// Examples of plant controlling.
// [Hint]
// > All reference-variables are implemented to ease monitoring of relevant variables.
FUNCTION_BLOCK FB_Plt_PlantControl EXTENDS FB_BA_View
VAR
   	{region 'Aggregates'}
		DmprSu_Open							: REFERENCE TO BOOL							REF= DmprSu.bOpen;
		DmprSu_Val							: REFERENCE TO REAL							REF= DmprSu.fActiveVal;
		DmprSu								: FB_TimerAggregateA						:= (iParent:=THIS^,					iLabel:=MyLabels.DmprSu);
		FanSu_Val							: REFERENCE TO UDINT						REF= FanSu.nActiveVal;
		FanSu								: FB_BA_AggregateM							:= (iParent:=THIS^,					iLabel:=MyLabels.FanSu);
			 
		DmprEx_Open							: REFERENCE TO BOOL							REF= DmprEx.bOpen;
		DmprEx_Val							: REFERENCE TO REAL							REF= DmprEx.fActiveVal;
		DmprEx								: FB_TimerAggregateA						:= (iParent:=THIS^,					iLabel:=MyLabels.DmprEx);
		FanEx_Val							: REFERENCE TO UDINT						REF= FanEx.nActiveVal;
		FanEx								: FB_BA_AggregateM							:= (iParent:=THIS^,					iLabel:=MyLabels.FanEx);
			 
		PreHtr_Proc							: REFERENCE TO BOOL							REF= PreHtr.Process.bActive;
		PreHtr_Val							: REFERENCE TO BOOL							REF= PreHtr.bActiveVal;
		PreHtr								: FB_ProcAggregateB							:= (iParent:=THIS^,					iLabel:=MyLabels.PreHtr,			Process:=(iLabel:=MyLabels.ProcPreRinse));
		Erc_Val								: REFERENCE TO BOOL							REF= Erc.bActiveVal;
		Erc									: FB_BA_AggregateB							:= (iParent:=THIS^,					iLabel:=MyLabels.Erc);
		Col_Val								: REFERENCE TO BOOL							REF= Col.bActiveVal;
		Col									: FB_BA_AggregateB							:= (iParent:=THIS^,					iLabel:=MyLabels.Col);
	{endregion}
	{region 'Plant'} 
		OpMode								: E_OpMod_AC								:= E_OpMod_AC.eOff;
		PlantCtrl_OpSta						: REFERENCE TO BOOL							REF= PlantCtrl.bOpSta;
		PlantCtrl_On						: REFERENCE TO BOOL							REF= PlantCtrl.bOn;
		PlantCtrl_PrVal						: REFERENCE TO UDINT						REF= PlantCtrl.nPresentValue;
		PlantCtrl_Step						: REFERENCE TO STRING						REF= PlantCtrl.sStep;
		PlantCtrl							: FB_BA_PlantCtrl := (
												iParent									:= THIS^,
												aOperationMode							:= [ E_OpMod_AC.eDisturb,			E_OpMod_AC.eSmokeExtract,		E_OpMod_AC.eOff,			E_OpMod_AC.eOn,				E_OpMod_AC.eNightCool ],
												aPriority								:= [ E_BA_Priority.eCritical,		E_BA_Priority.eLifeSafety,		E_BA_Priority.eProgram,		E_BA_Priority.eProgram,		E_BA_Priority.eProgram ],
												aAggregates := [(
													iReference							:= DmprSu,
													aOpMode								:= [ 0,								100,							0,							100,						100 ]
												), (
													iReference							:= DmprEx,
													aOpMode								:= [ 0,								100,							0,							100,						100 ]
												), (
													iReference							:= PreHtr,
													aOpMode								:= [ E_OpMod_Binary.eOff,			E_OpMod_Binary.eOn,				E_OpMod_Binary.eOff,		E_OpMod_Binary.eOn,			E_OpMod_Binary.eOff ],
													bWaitForProcesses					:= TRUE
												), (
													iReference							:= Erc,
													aOpMode								:= [ E_OpMod_Binary.eOff,			E_OpMod_Binary.eOn,				E_OpMod_Binary.eOff,		E_OpMod_Binary.eOn,			E_OpMod_Binary.eOff ]
												), (
													iReference							:= Col,
													aOpMode								:= [ E_OpMod_Binary.eOff,			E_OpMod_Binary.eOn,				E_OpMod_Binary.eOff,		E_OpMod_Binary.eOn,			E_OpMod_Binary.eOff ]
												), (
													iReference							:= FanSu,
													aOpMode								:= [ E_OpMod_Step2.eOff,			E_OpMod_Step2.eStep2,			E_OpMod_Step2.eOff,			E_OpMod_Step2.eStep1,		E_OpMod_Step2.eStep2 ],
													tDelayStepDown						:= T#0S,
													tDelayStepUp						:= T#5S
												), (
													iReference							:= FanEx,
													aOpMode								:= [ E_OpMod_Step2.eOff,			E_OpMod_Step2.eStep2,			E_OpMod_Step2.eOff,			E_OpMod_Step2.eStep1,		E_OpMod_Step2.eStep2 ],
													tDelayStepDown						:= T#5S,
													tDelayStepUp						:= T#0S
												)]
											);
	{endregion}
END_VAR

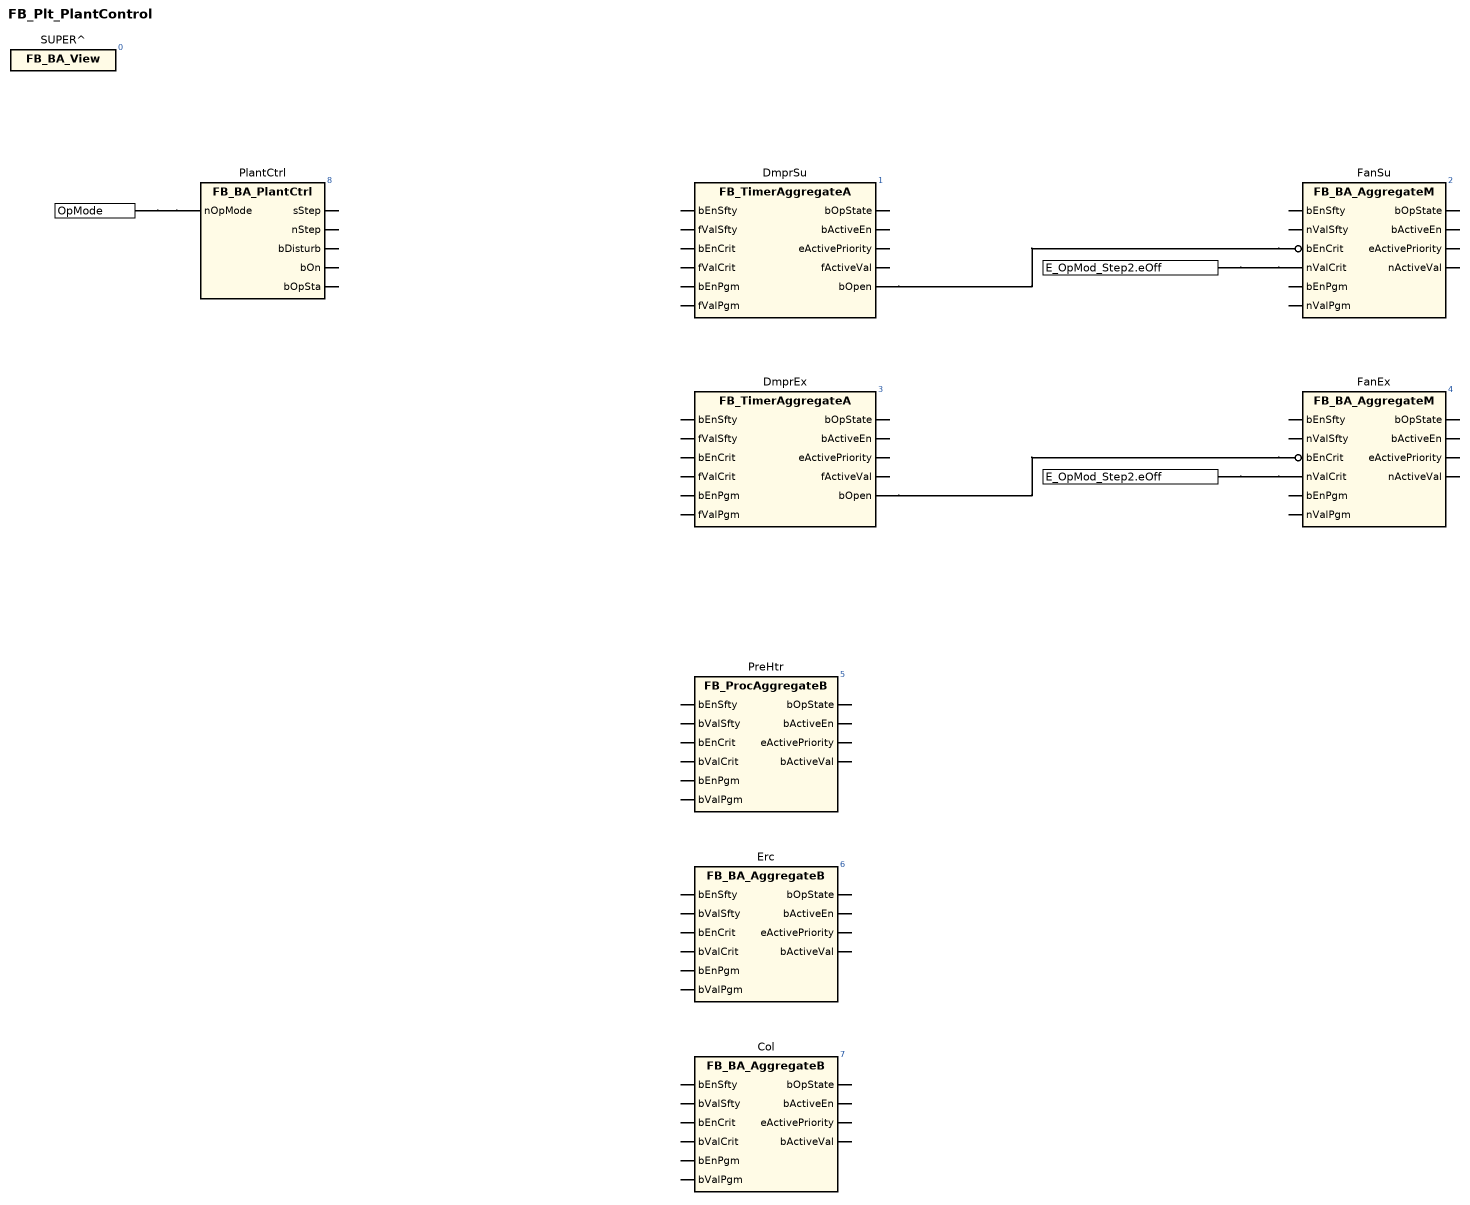
SUPER^(); // FB_BA_View
DmprSu(); // FB_TimerAggregateA
FanSu(bEnCrit := NOT DmprSu.bOpen, nValCrit := E_OpMod_Step2.eOff); // FB_BA_AggregateM
DmprEx(); // FB_TimerAggregateA
FanEx(bEnCrit := NOT DmprEx.bOpen, nValCrit := E_OpMod_Step2.eOff); // FB_BA_AggregateM
PreHtr(); // FB_ProcAggregateB
Erc(); // FB_BA_AggregateB
Col(); // FB_BA_AggregateB
PlantCtrl(nOpMode := OpMode); // FB_BA_PlantCtrl

// Alternative to initialization at FB-Declararion:
// > Initialization-Methods in "FB_init"
METHOD FB_init : BOOL
VAR_INPUT
	bInitRetains : BOOL; // if TRUE, the retain variables are initialized (warm start / cold start)
	bInCopyCode : BOOL;  // if TRUE, the instance afterwards gets moved into the copy code (online change)
END_VAR
PlantCtrl.Clear();

// Add plant operations modes:
PlantCtrl.AddOperationMode(E_OpMod_AC.eDisturb,			E_BA_Priority.eCritical);
PlantCtrl.AddOperationMode(E_OpMod_AC.eSmokeExtract,	E_BA_Priority.eLifeSafety);
PlantCtrl.AddOperationMode(E_OpMod_AC.eOff,				E_BA_Priority.eProgram);
PlantCtrl.AddOperationMode(E_OpMod_AC.eOn,				E_BA_Priority.eProgram);
PlantCtrl.AddOperationMode(E_OpMod_AC.eNightCool,		E_BA_Priority.eProgram);

// Add aggregates:
PlantCtrl.AddAggregate(DmprSu,	FALSE,	FALSE,	T#0S,	T#0S);
PlantCtrl.AddAggregate(DmprEx,	FALSE,	FALSE,	T#0S,	T#0S);
PlantCtrl.AddAggregate(PreHtr,	TRUE,	FALSE,	T#0S,	T#0S);
PlantCtrl.AddAggregate(Erc,		FALSE,	FALSE,	T#0S,	T#0S);
PlantCtrl.AddAggregate(Col,		FALSE,	FALSE,	T#0S,	T#0S);
PlantCtrl.AddAggregate(FanSu,	FALSE,	FALSE,	T#0S,	T#5S);
PlantCtrl.AddAggregate(FanEx,	FALSE,	FALSE,	T#5S,	T#0S);

// Apply aggregate operation modes dependant on corresponding plant operation modes:
PlantCtrl.AssignAggregate4x(E_OpMod_AC.eDisturb,		DmprSu, TO_UDINT(0),					FanSu, TO_UDINT(E_OpMod_Step2.eOff),		DmprEx, TO_UDINT(0),					FanEx, TO_UDINT(E_OpMod_Step2.eOff));
PlantCtrl.AssignAggregate4x(E_OpMod_AC.eSmokeExtract,	DmprSu, TO_UDINT(100),					FanSu, TO_UDINT(E_OpMod_Step2.eStep2),		DmprEx, TO_UDINT(100),					FanEx, TO_UDINT(E_OpMod_Step2.eStep2));
PlantCtrl.AssignAggregate4x(E_OpMod_AC.eOff,			DmprSu, TO_UDINT(0),					FanSu, TO_UDINT(E_OpMod_Step2.eOff),		DmprEx, TO_UDINT(0),					FanEx, TO_UDINT(E_OpMod_Step2.eOff));
PlantCtrl.AssignAggregate4x(E_OpMod_AC.eOn,				DmprSu, TO_UDINT(100),					FanSu, TO_UDINT(E_OpMod_Step2.eStep1),		DmprEx, TO_UDINT(100),					FanEx, TO_UDINT(E_OpMod_Step2.eStep1));
PlantCtrl.AssignAggregate4x(E_OpMod_AC.eNightCool,		DmprSu, TO_UDINT(100),					FanSu, TO_UDINT(E_OpMod_Step2.eStep2),		DmprEx, TO_UDINT(100),					FanEx, TO_UDINT(E_OpMod_Step2.eStep2));

PlantCtrl.AssignAggregate3x(E_OpMod_AC.eDisturb,		PreHtr, TO_UDINT(E_OpMod_Binary.eOff),	Erc, TO_UDINT(E_OpMod_Binary.eOff),			Col, TO_UDINT(E_OpMod_Binary.eOff));
PlantCtrl.AssignAggregate3x(E_OpMod_AC.eSmokeExtract,	PreHtr, TO_UDINT(E_OpMod_Binary.eOn),	Erc, TO_UDINT(E_OpMod_Binary.eOn),			Col, TO_UDINT(E_OpMod_Binary.eOn));
PlantCtrl.AssignAggregate3x(E_OpMod_AC.eOff,			PreHtr, TO_UDINT(E_OpMod_Binary.eOff),	Erc, TO_UDINT(E_OpMod_Binary.eOff),			Col, TO_UDINT(E_OpMod_Binary.eOff));
PlantCtrl.AssignAggregate3x(E_OpMod_AC.eOn,				PreHtr, TO_UDINT(E_OpMod_Binary.eOn),	Erc, TO_UDINT(E_OpMod_Binary.eOn),			Col, TO_UDINT(E_OpMod_Binary.eOn));
PlantCtrl.AssignAggregate3x(E_OpMod_AC.eNightCool,		PreHtr, TO_UDINT(E_OpMod_Binary.eOff),	Erc, TO_UDINT(E_OpMod_Binary.eOff),			Col, TO_UDINT(E_OpMod_Binary.eOff));
END_METHOD

END_FUNCTION_BLOCK

(* stored: Version 1.1.0.1, ProductVersion 3.1.4024.10
   POU FB_Plt_PlantControl: Id {a9ce6917-417d-453a-ad36-bec8d12e7989}, SpecialFunc None
   Method FB_init: Id {1aeb9bc9-bf4d-4c6e-80f8-3e27167b97f4} *)
